FUNCTION Count_to_MeasureUnits : REAL
VAR_INPUT
	iValue_in	: INT; 
	iHigh		: REAL;
	iLow		: REAL;
END_VAR
VAR
END_VAR

Count_to_MeasureUnits := ((iHigh - iLow) / 32767.0) * INT_TO_REAL(iValue_In) + iLow;

END_FUNCTION

(* stored: Version 1.1.0.1, ProductVersion 3.1.4024.12
   POU Count_to_MeasureUnits: Id {1e75b0e8-fced-4942-bada-b0161c2e5412}, SpecialFunc None *)
